TYPE TYP_HW_EL6001 :
STRUCT
	In : TYP_HW_EL6001_IN;
	Out : TYP_HW_EL6001_OUT;
END_STRUCT
END_TYPE

(* stored: Version 1.1.0.1, ProductVersion 3.1.4024.12
   DUT TYP_HW_EL6001: Id {091a51fd-9a83-4bf4-a690-cc6a9c96af80} *)
